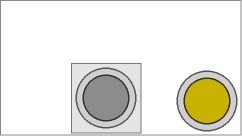
VISUALIZATION Visualization_Carbid  // 242x136
    Lamp1 (172,66 70x70), variable: GVL_Carbid.Lamp, style: Lamp-Lamp1-Yellow
    PushSwitch (71,63 70x70), variable: GVL_Carbid.Button, behaviour: TOGGLE, style: Switch-PushSwitch-Gray
END_VISUALIZATION

(* stored: Version 1.1.0.1, ProductVersion 3.1.4024.12
   Visu Visualization_Carbid: Id {2d3925e2-05c9-4339-99be-acef35c2da14} *)
